(* Logix 5000 project; controller ARS14002_PLC vendor 1 type 14 code 218 rev 30.11; software revision 30.01; part 10 of 13 *)
(* tags used below, declared in another part *)
   DERIME_EMPTY : BOOL;
   DERIME_EMPTY_ALARM : BOOL;
   DERIME_EMPTY_HOLD_TMR : TIMER;
   DERIME_FILL : BOOL;
   DERIME_FULL : BOOL;
   DERIME_FULL_ALARM : BOOL;
   DERIME_FULL_HOLD_TMR : TIMER;
   DERIME_SPH : REAL;
   DERIME_SPL : REAL;
   DERIME_VENT : BOOL;
   ARS_DERIME_AUTO : BOOL;
   AT2_PLANT_ATOMIZING : BOOL;
   AT3_PLANT_ATOMIZING : BOOL;
   BLOWBACK_PRESS_SPH : REAL;
   BLOWBACK_PRESS_SPL : REAL;
   BLOWBACK_PRESS_UNSAFE : REAL;
   DERIME_HOLD : BOOL;
   DERIME_HP_CYCLE : BOOL;
   DERIME_HP_SPH : REAL;   // SETPOINT FOR VALVES BESIDES FCV-202
   DERIME_HP_SPL : REAL;   // SETPOIT FOR VALVES BESIDES FCV-202
   FCV_202 : CM_AO_VLV;
   FCV_202_BLOWBACK_POS : REAL;
   FCV_504_SP_Standby : REAL;
   FCV_504_SP_Standby_AR : REAL;
   FCV_504_SP_Standby_FRONT_END : REAL;
   FIRST_SCAN_BIT : BOOL;
   FVR_800C_RUNNING : BOOL;
   FVR_800D_RUNNING : BOOL;
   MTR_550 : CM_DO_FVNR;
   PDT_1101A : CM_AI_SCL_ALT;
   PIDE_101A : PID_ENHANCED;
   PIDE_101B : PID_ENHANCED;
   PIDE_101C : PID_ENHANCED;
   PIDE_102A : PID_ENHANCED;
   PIDE_102B : PID_ENHANCED;
   PIDE_102C : PID_ENHANCED;
   PIDE_202 : PID_ENHANCED;
   PIDE_204 : PID_ENHANCED;
   PIDE_207 : PID_ENHANCED;
   PIDE_504 : PID_ENHANCED;
   PIDE_504_COLDBOX_IGAIN : REAL;
   PIDE_504_COLDBOX_PGAIN : REAL;
   PIDE_504_FRONT_END_CONTROL : BOOL;
   PIDE_504_FRONT_END_IGAIN : REAL;
   PIDE_504_FRONT_END_PGAIN : REAL;
   PIDE_504_MODE : BOOL;   // 0 = Argon (PT-601) 1 = N2 (PT-603)
   PIDE_504_PVCHANGE1 : BOOL;
   PIDE_504_PVCHANGE2 : BOOL;
   PIDE_504_PVCHANGE3 : BOOL;
   PIDE_504_RESET : BOOL;
   PIDE_603 : PID_ENHANCED;
   PILOT_PLANT_ATOMIZING : BOOL;
   PT_1003 : CM_AI_SCL;
   PT_1101A : CM_AI_SCL;
   PT_1301A : CM_AI_SCL;
   PT_1301B : CM_AI_SCL;
   PT_201 : CM_AI_SCL;
   PT_601 : CM_AI_SCL;
   PT_603 : CM_AI_SCL;
   PT_701 : CM_AI_SCL;
   PT_806 : CM_AI_SCL;
   PWHMI_OutletValveStatus : BOOL;
   SV_1005_SPH : INT;
   SV_1005_SPL : INT;
   SV_1005X : CM_DO_GENERIC;
   SV_101AF : CM_DO_GENERIC;
   SV_101BF : CM_DO_GENERIC;
   SV_101CF : CM_DO_GENERIC;
   SV_102AF : CM_DO_GENERIC;
   SV_102BF : CM_DO_GENERIC;
   SV_102CF : CM_DO_GENERIC;
   SV_1104A : CM_DO_GENERIC;
   SV_1109AX : CM_DO_GENERIC;
   SV_1304A : CM_DO_GENERIC;
   SV_1304B : CM_DO_GENERIC;
   SV_1309AX : CM_DO_GENERIC;
   SV_1309BX : CM_DO_GENERIC;
   SV_202F : CM_DO_GENERIC;
   SV_204F : CM_DO_GENERIC;
   SV_207F : CM_DO_GENERIC;
   SV_504F : CM_DO_GENERIC;
   TK_1100A_Low : BOOL;
   TK_1100A_LOW_DLA_TMR : TIMER;
   TK_1100A_Low_SPH : REAL;
   TK_1100A_Low_SPL : REAL;
   TK_1100A_Low_Warning : BOOL;
   TK_1100A_LOW_WARNING_DLA_TMR : TIMER;
   TK_1100A_Low_WARNING_SPH : REAL;
   TK_1100A_Low_WARNING_SPL : REAL;
   TK_1100A_PBC_Pressure_SPH : INT;
   TK_1100A_PBC_Pressure_SPL : INT;
   TK_1100A_Vent_Closed_TMR : TIMER;
   TK_1100A_Vent_Open_TMR : TIMER;
   TK_1100A_Vent_Pressure_SPH : INT;
   TK_1100A_Vent_Pressure_SPL : INT;
   TK_1300A_PBC_Pressure_SPH : INT;
   TK_1300A_PBC_Pressure_SPL : INT;
   TK_1300A_Vent_Closed_TMR : TIMER;
   TK_1300A_Vent_Open_TMR : TIMER;
   TK_1300A_Vent_Pressure_SPH : INT;
   TK_1300A_Vent_Pressure_SPL : INT;
   TK_1300B_Vent_Closed_TMR : TIMER;
   TK_1300B_Vent_Open_TMR : TIMER;
   XV_623 : CM_DO_VLV;
   XV_623_FILL_MODE : BOOL;   // (0=Manual, 1=Auto)
   XV_623_SPH : INT;
   XV_623_SPL : INT;
   XV_801A : CM_DO_VLV;
   XV_801B : CM_DO_VLV;
   XV_801C : CM_DO_VLV;
   XV_801D : CM_DO_VLV;
   XV_806 : CM_DO_VLV;
(* MainProgram, continued *)

ROUTINE _310_TK_1100A   (* ladder *)
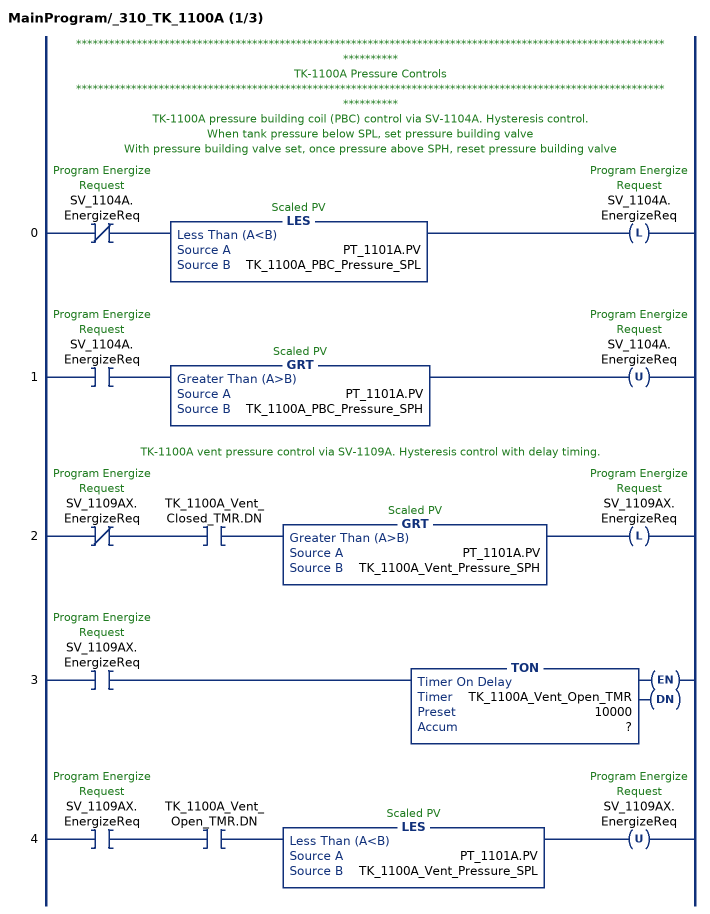
   // *********************************************************************************************************************
   // TK-1100A Pressure Controls
   // *********************************************************************************************************************
   // TK-1100A pressure building coil (PBC) control via SV-1104A. Hysteresis control.
   // When tank pressure below SPL, set pressure building valve
   // With pressure building valve set, once pressure above SPH, reset pressure building valve
   0: XIO(SV_1104A.EnergizeReq)LES(PT_1101A.PV,TK_1100A_PBC_Pressure_SPL)OTL(SV_1104A.EnergizeReq);
   1: XIC(SV_1104A.EnergizeReq)GRT(PT_1101A.PV,TK_1100A_PBC_Pressure_SPH)OTU(SV_1104A.EnergizeReq);
   // TK-1100A vent pressure control via SV-1109A. Hysteresis control with delay timing.
   2: XIO(SV_1109AX.EnergizeReq)XIC(TK_1100A_Vent_Closed_TMR.DN)GRT(PT_1101A.PV,TK_1100A_Vent_Pressure_SPH)OTL(SV_1109AX.EnergizeReq);
   3: XIC(SV_1109AX.EnergizeReq)TON(TK_1100A_Vent_Open_TMR,?,?);
   4: XIC(SV_1109AX.EnergizeReq)XIC(TK_1100A_Vent_Open_TMR.DN)LES(PT_1101A.PV,TK_1100A_Vent_Pressure_SPL)OTU(SV_1109AX.EnergizeReq);
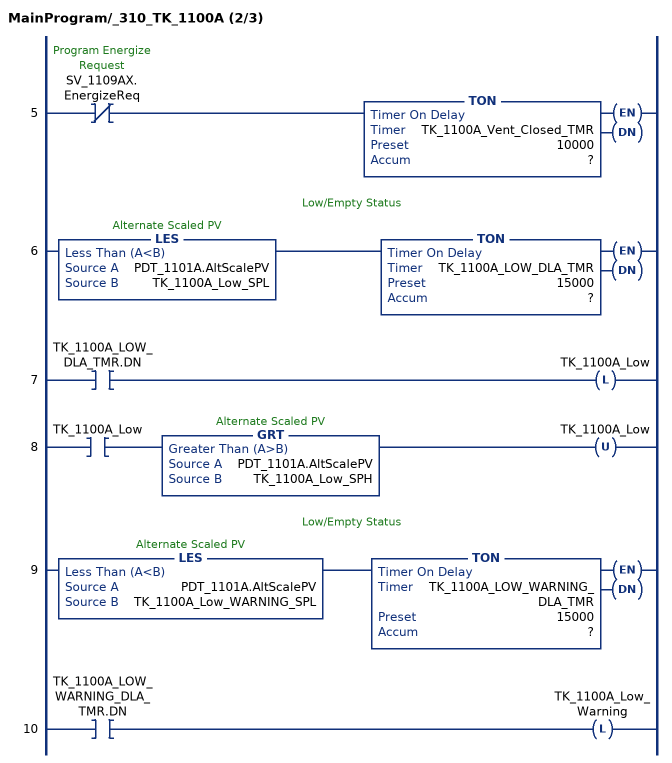
   5: XIO(SV_1109AX.EnergizeReq)TON(TK_1100A_Vent_Closed_TMR,?,?);
   // Low/Empty Status
   6: LES(PDT_1101A.AltScalePV,TK_1100A_Low_SPL)TON(TK_1100A_LOW_DLA_TMR,?,?);
   7: XIC(TK_1100A_LOW_DLA_TMR.DN)OTL(TK_1100A_Low);
   8: XIC(TK_1100A_Low)GRT(PDT_1101A.AltScalePV,TK_1100A_Low_SPH)OTU(TK_1100A_Low);
   // Low/Empty Status
   9: LES(PDT_1101A.AltScalePV,TK_1100A_Low_WARNING_SPL)TON(TK_1100A_LOW_WARNING_DLA_TMR,?,?);
   10: XIC(TK_1100A_LOW_WARNING_DLA_TMR.DN)OTL(TK_1100A_Low_Warning);
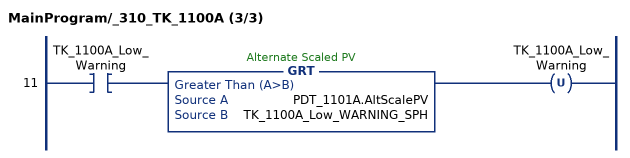
   11: XIC(TK_1100A_Low_Warning)GRT(PDT_1101A.AltScalePV,TK_1100A_Low_WARNING_SPH)OTU(TK_1100A_Low_Warning);
END_ROUTINE

ROUTINE _311A_TK_1300A   (* ladder *)
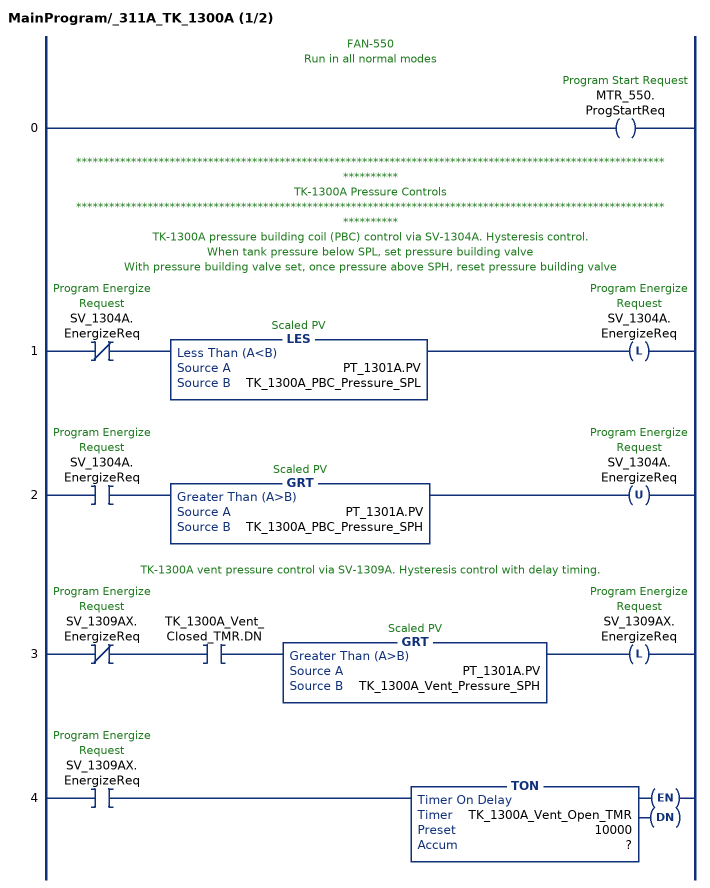
   // FAN-550
   // Run in all normal modes
   0: OTE(MTR_550.ProgStartReq);
   // *********************************************************************************************************************
   // TK-1300A Pressure Controls
   // *********************************************************************************************************************
   // TK-1300A pressure building coil (PBC) control via SV-1304A. Hysteresis control.
   // When tank pressure below SPL, set pressure building valve
   // With pressure building valve set, once pressure above SPH, reset pressure building valve
   1: XIO(SV_1304A.EnergizeReq)LES(PT_1301A.PV,TK_1300A_PBC_Pressure_SPL)OTL(SV_1304A.EnergizeReq);
   2: XIC(SV_1304A.EnergizeReq)GRT(PT_1301A.PV,TK_1300A_PBC_Pressure_SPH)OTU(SV_1304A.EnergizeReq);
   // TK-1300A vent pressure control via SV-1309A. Hysteresis control with delay timing.
   3: XIO(SV_1309AX.EnergizeReq)XIC(TK_1300A_Vent_Closed_TMR.DN)GRT(PT_1301A.PV,TK_1300A_Vent_Pressure_SPH)OTL(SV_1309AX.EnergizeReq);
   4: XIC(SV_1309AX.EnergizeReq)TON(TK_1300A_Vent_Open_TMR,?,?);
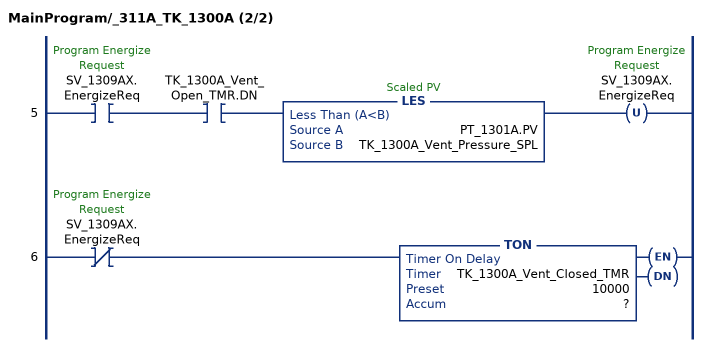
   5: XIC(SV_1309AX.EnergizeReq)XIC(TK_1300A_Vent_Open_TMR.DN)LES(PT_1301A.PV,TK_1300A_Vent_Pressure_SPL)OTU(SV_1309AX.EnergizeReq);
   6: XIO(SV_1309AX.EnergizeReq)TON(TK_1300A_Vent_Closed_TMR,?,?);
END_ROUTINE

ROUTINE _311B_TK_1300B   (* ladder *)
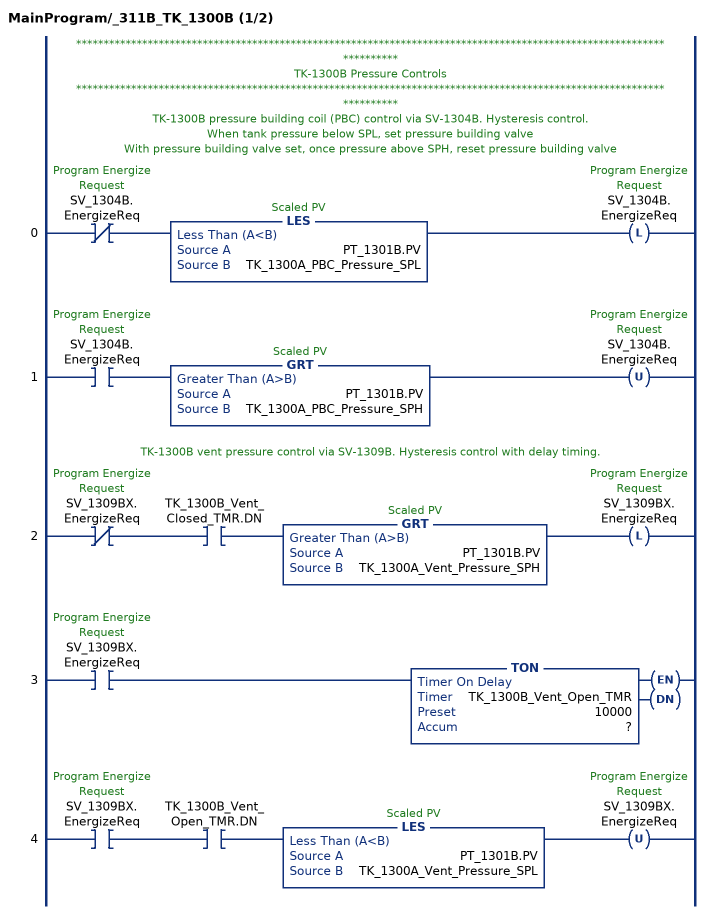
   // *********************************************************************************************************************
   // TK-1300B Pressure Controls
   // *********************************************************************************************************************
   // TK-1300B pressure building coil (PBC) control via SV-1304B. Hysteresis control.
   // When tank pressure below SPL, set pressure building valve
   // With pressure building valve set, once pressure above SPH, reset pressure building valve
   0: XIO(SV_1304B.EnergizeReq)LES(PT_1301B.PV,TK_1300A_PBC_Pressure_SPL)OTL(SV_1304B.EnergizeReq);
   1: XIC(SV_1304B.EnergizeReq)GRT(PT_1301B.PV,TK_1300A_PBC_Pressure_SPH)OTU(SV_1304B.EnergizeReq);
   // TK-1300B vent pressure control via SV-1309B. Hysteresis control with delay timing.
   2: XIO(SV_1309BX.EnergizeReq)XIC(TK_1300B_Vent_Closed_TMR.DN)GRT(PT_1301B.PV,TK_1300A_Vent_Pressure_SPH)OTL(SV_1309BX.EnergizeReq);
   3: XIC(SV_1309BX.EnergizeReq)TON(TK_1300B_Vent_Open_TMR,?,?);
   4: XIC(SV_1309BX.EnergizeReq)XIC(TK_1300B_Vent_Open_TMR.DN)LES(PT_1301B.PV,TK_1300A_Vent_Pressure_SPL)OTU(SV_1309BX.EnergizeReq);
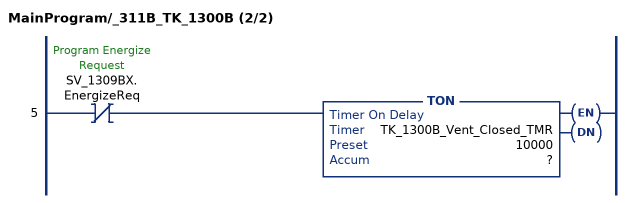
   5: XIO(SV_1309BX.EnergizeReq)TON(TK_1300B_Vent_Closed_TMR,?,?);
END_ROUTINE

ROUTINE _312_Misc_Hysteresis   (* ladder *)
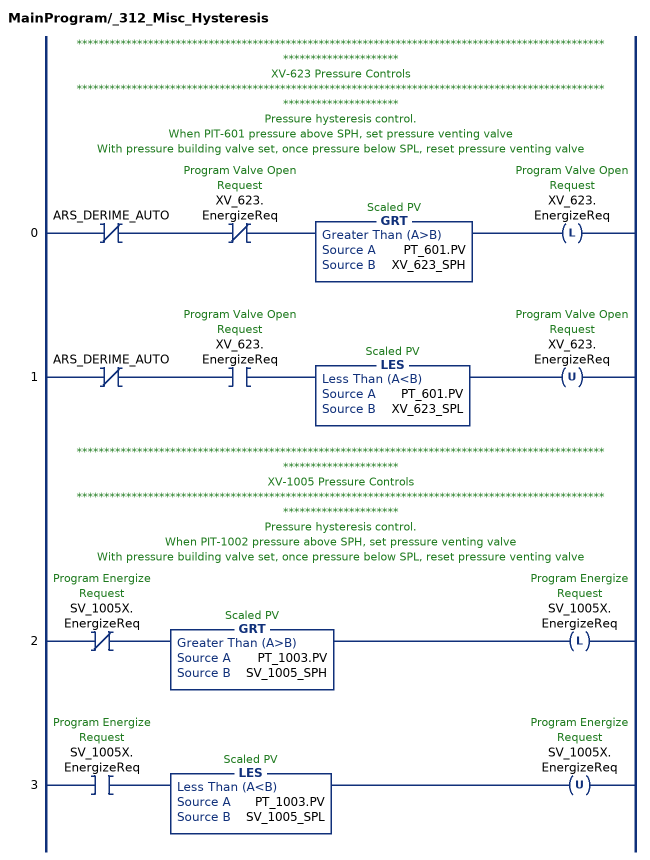
   // *********************************************************************************************************************
   // XV-623 Pressure Controls
   // *********************************************************************************************************************
   // Pressure hysteresis control.
   // When PIT-601 pressure above SPH, set pressure venting valve
   // With pressure building valve set, once pressure below SPL, reset pressure venting valve
   0: XIO(ARS_DERIME_AUTO)XIO(XV_623.EnergizeReq)GRT(PT_601.PV,XV_623_SPH)OTL(XV_623.EnergizeReq);
   1: XIO(ARS_DERIME_AUTO)XIC(XV_623.EnergizeReq)LES(PT_601.PV,XV_623_SPL)OTU(XV_623.EnergizeReq);
   // *********************************************************************************************************************
   // XV-1005 Pressure Controls
   // *********************************************************************************************************************
   // Pressure hysteresis control.
   // When PIT-1002 pressure above SPH, set pressure venting valve
   // With pressure building valve set, once pressure below SPL, reset pressure venting valve
   2: XIO(SV_1005X.EnergizeReq)GRT(PT_1003.PV,SV_1005_SPH)OTL(SV_1005X.EnergizeReq);
   3: XIC(SV_1005X.EnergizeReq)LES(PT_1003.PV,SV_1005_SPL)OTU(SV_1005X.EnergizeReq);
END_ROUTINE

ROUTINE _313_Derime   (* ladder *)
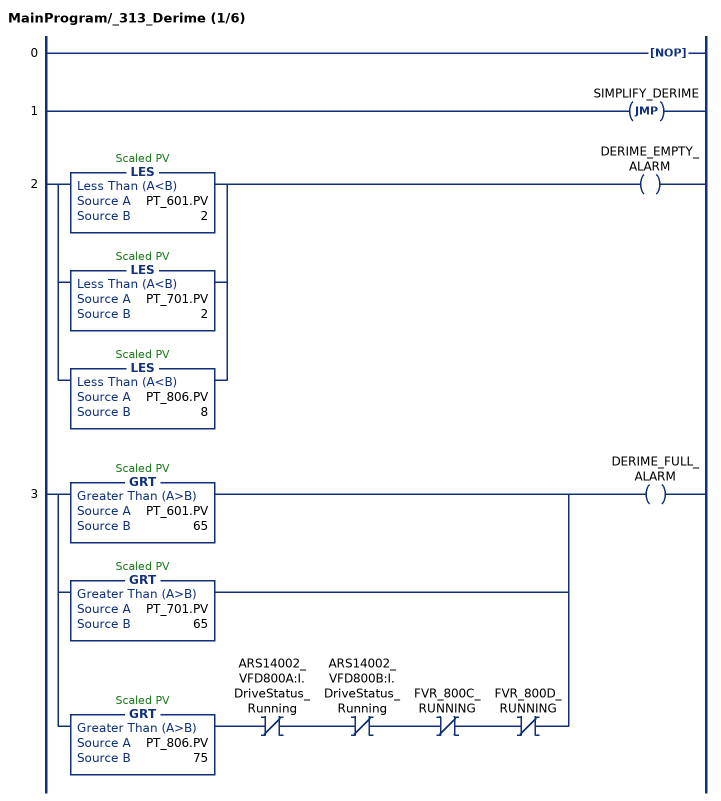
   0: NOP();
   1: JMP(SIMPLIFY_DERIME);
   2: [LES(PT_601.PV,2) ,LES(PT_701.PV,2) ,LES(PT_806.PV,8) ]OTE(DERIME_EMPTY_ALARM);
   3: [GRT(PT_601.PV,65) ,GRT(PT_701.PV,65) ,GRT(PT_806.PV,75) XIO(ARS14002_VFD800A:I.DriveStatus_Running) XIO(ARS14002_VFD800B:I.DriveStatus_Running) XIO(FVR_800C_RUNNING) XIO(FVR_800D_RUNNING) ]OTE(DERIME_FULL_ALARM);
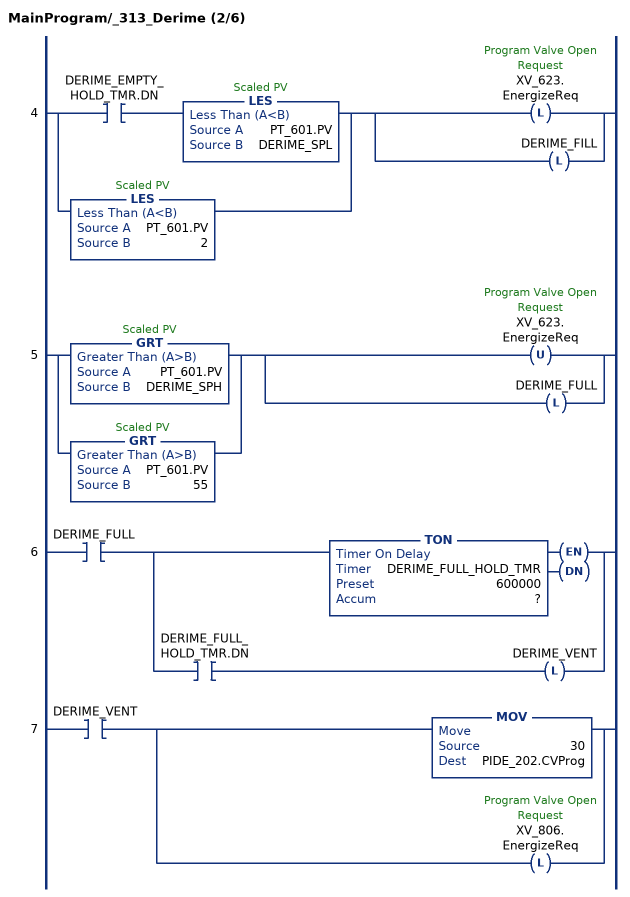
   4: [XIC(DERIME_EMPTY_HOLD_TMR.DN) LES(PT_601.PV,DERIME_SPL) ,LES(PT_601.PV,2) ][OTL(XV_623.EnergizeReq) ,OTL(DERIME_FILL) ];
   5: [GRT(PT_601.PV,DERIME_SPH) ,GRT(PT_601.PV,55) ][OTU(XV_623.EnergizeReq) ,OTL(DERIME_FULL) ];
   6: XIC(DERIME_FULL)[TON(DERIME_FULL_HOLD_TMR,?,?) ,XIC(DERIME_FULL_HOLD_TMR.DN) OTL(DERIME_VENT) ];
   7: XIC(DERIME_VENT)[MOV(30,PIDE_202.CVProg) ,OTL(XV_806.EnergizeReq) ];
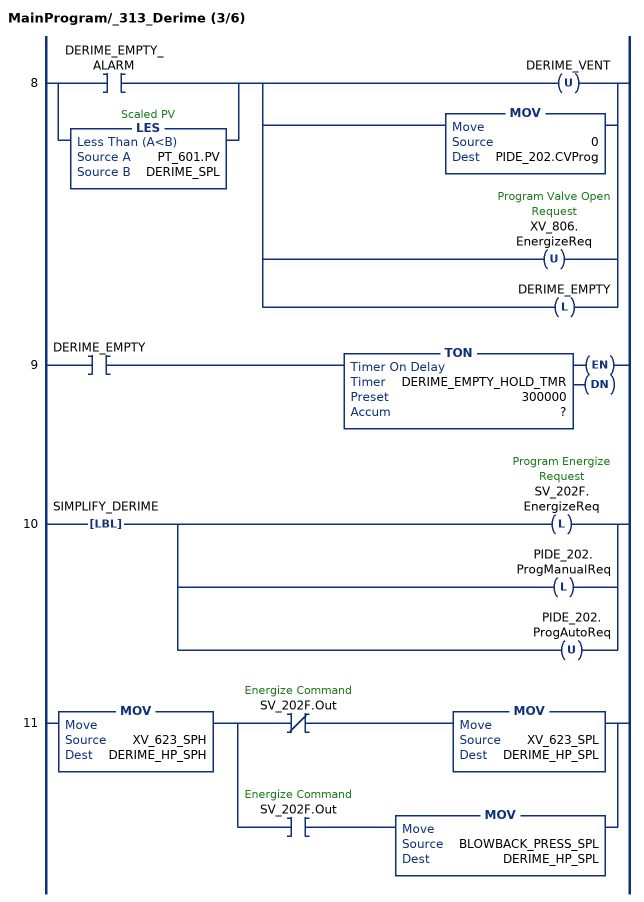
   8: [XIC(DERIME_EMPTY_ALARM) ,LES(PT_601.PV,DERIME_SPL) ][OTU(DERIME_VENT) ,MOV(0,PIDE_202.CVProg) ,OTU(XV_806.EnergizeReq) ,OTL(DERIME_EMPTY) ];
   9: XIC(DERIME_EMPTY)TON(DERIME_EMPTY_HOLD_TMR,?,?);
   10: LBL(SIMPLIFY_DERIME)[OTL(SV_202F.EnergizeReq) ,OTL(PIDE_202.ProgManualReq) ,OTU(PIDE_202.ProgAutoReq) ];
   11: MOV(XV_623_SPH,DERIME_HP_SPH)[XIO(SV_202F.Out) MOV(XV_623_SPL,DERIME_HP_SPL) ,XIC(SV_202F.Out) MOV(BLOWBACK_PRESS_SPL,DERIME_HP_SPL) ];
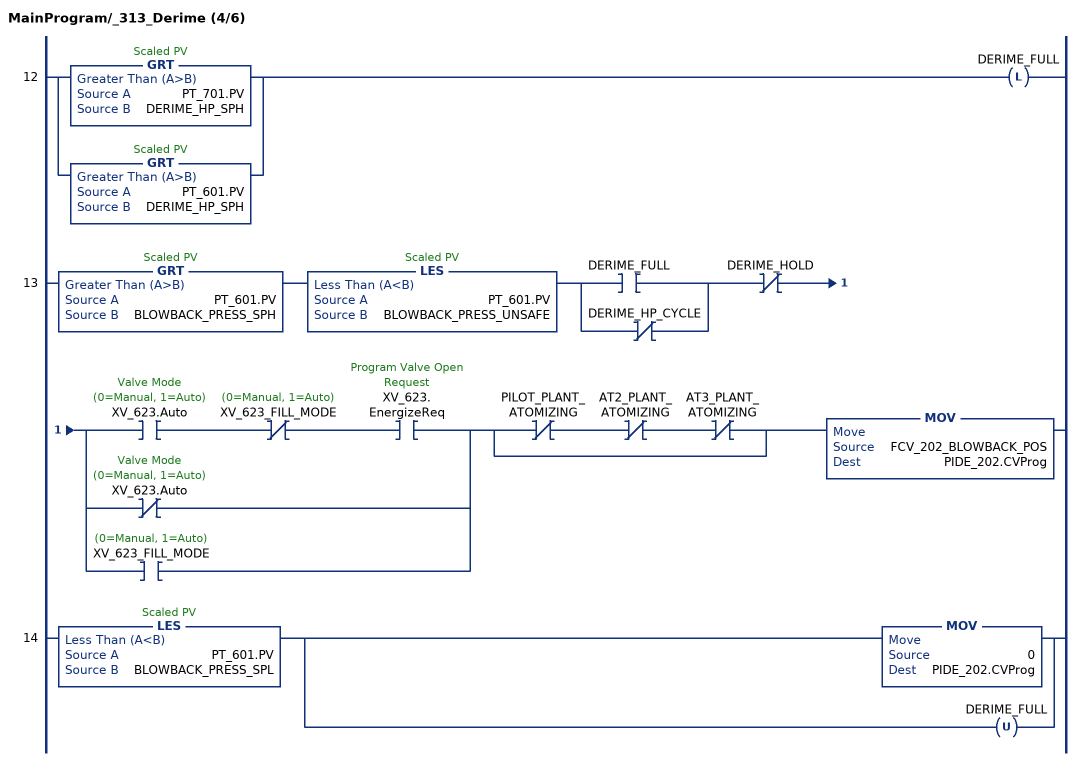
   12: [GRT(PT_701.PV,DERIME_HP_SPH) ,GRT(PT_601.PV,DERIME_HP_SPH) ]OTL(DERIME_FULL);
   13: GRT(PT_601.PV,BLOWBACK_PRESS_SPH)LES(PT_601.PV,BLOWBACK_PRESS_UNSAFE)[XIC(DERIME_FULL) ,XIO(DERIME_HP_CYCLE) ]XIO(DERIME_HOLD)[XIC(XV_623.Auto) XIO(XV_623_FILL_MODE) XIC(XV_623.EnergizeReq) ,XIO(XV_623.Auto) ,XIC(XV_623_FILL_MODE) ][XIO(PILOT_PLANT_ATOMIZING) XIO(AT2_PLANT_ATOMIZING) XIO(AT3_PLANT_ATOMIZING) ,]MOV(FCV_202_BLOWBACK_POS,PIDE_202.CVProg);
   14: LES(PT_601.PV,BLOWBACK_PRESS_SPL)[MOV(0,PIDE_202.CVProg) ,OTU(DERIME_FULL) ];
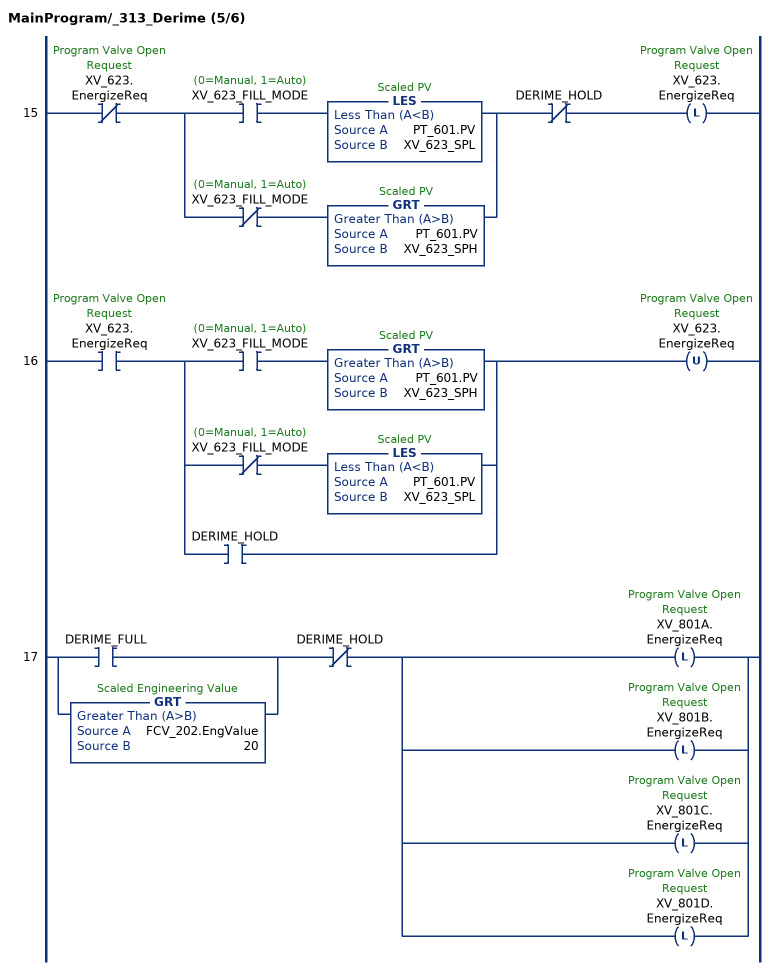
   15: XIO(XV_623.EnergizeReq)[XIC(XV_623_FILL_MODE) LES(PT_601.PV,XV_623_SPL) ,XIO(XV_623_FILL_MODE) GRT(PT_601.PV,XV_623_SPH) ]XIO(DERIME_HOLD)OTL(XV_623.EnergizeReq);
   16: XIC(XV_623.EnergizeReq)[XIC(XV_623_FILL_MODE) GRT(PT_601.PV,XV_623_SPH) ,XIO(XV_623_FILL_MODE) LES(PT_601.PV,XV_623_SPL) ,XIC(DERIME_HOLD) ]OTU(XV_623.EnergizeReq);
   17: [XIC(DERIME_FULL) ,GRT(FCV_202.EngValue,20) ]XIO(DERIME_HOLD)[OTL(XV_801A.EnergizeReq) ,OTL(XV_801B.EnergizeReq) ,OTL(XV_801C.EnergizeReq) ,OTL(XV_801D.EnergizeReq) ];
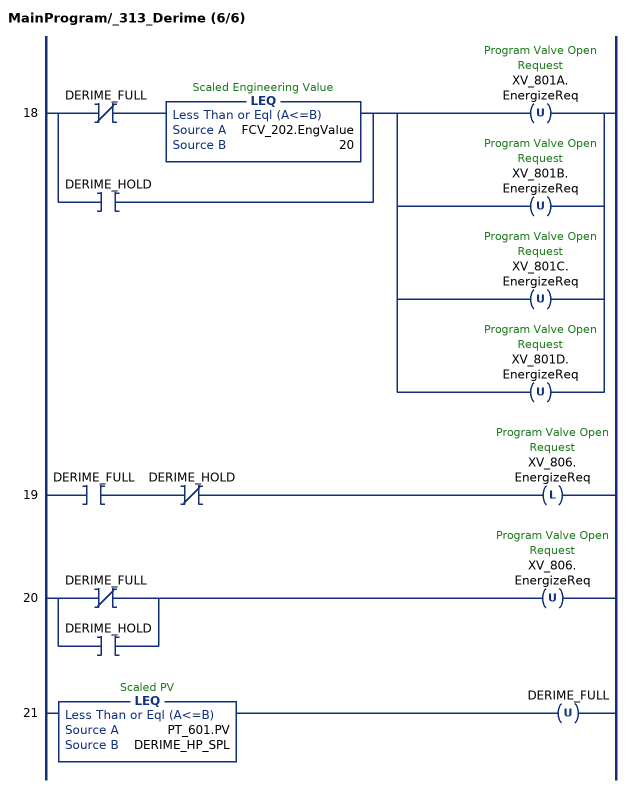
   18: [XIO(DERIME_FULL) LEQ(FCV_202.EngValue,20) ,XIC(DERIME_HOLD) ][OTU(XV_801A.EnergizeReq) ,OTU(XV_801B.EnergizeReq) ,OTU(XV_801C.EnergizeReq) ,OTU(XV_801D.EnergizeReq) ];
   19: XIC(DERIME_FULL)XIO(DERIME_HOLD)OTL(XV_806.EnergizeReq);
   20: [XIO(DERIME_FULL) ,XIC(DERIME_HOLD) ]OTU(XV_806.EnergizeReq);
   21: LEQ(PT_601.PV,DERIME_HP_SPL)OTU(DERIME_FULL);
END_ROUTINE

ROUTINE _40_Process_PID_Misc   (* ladder *)
// PID state transition logic
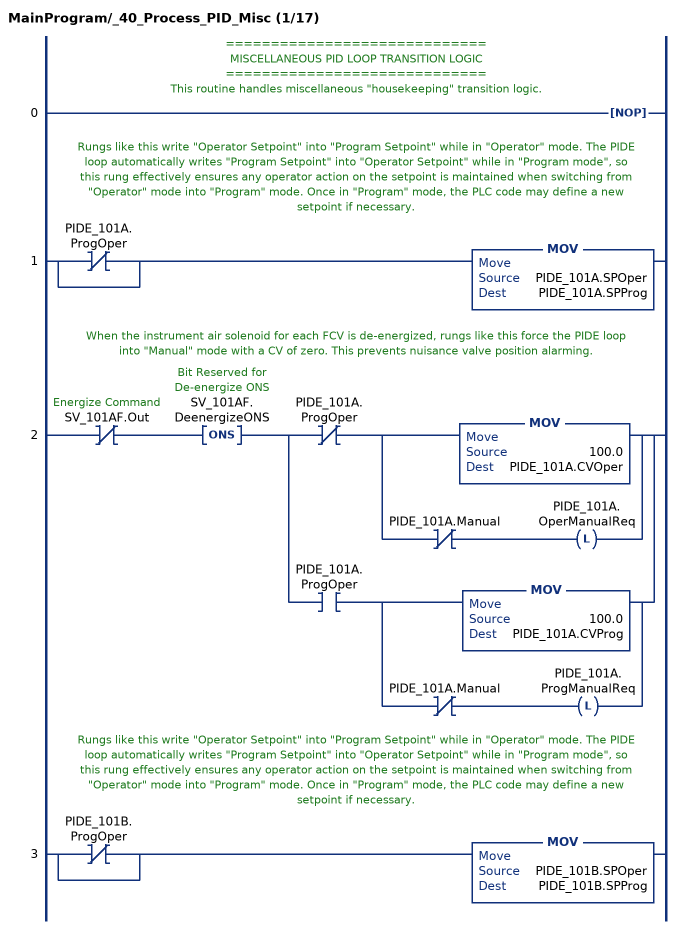
   // =============================
   // MISCELLANEOUS PID LOOP TRANSITION LOGIC
   // =============================
   //  This routine handles miscellaneous "housekeeping" transition logic.
   0: NOP();
   // Rungs like this write "Operator Setpoint" into "Program Setpoint" while in "Operator" mode. The PIDE loop automatically writes "Program Setpoint" into "Operator Setpoint" while in "Program mode", so this rung effectively ensures any operator action on the setpoint is maintained when switching from "Operator" mode into "Program" mode. Once in "Program" mode, the PLC code may define a new setpoint if necessary.
   1: [XIO(PIDE_101A.ProgOper) ,]MOV(PIDE_101A.SPOper,PIDE_101A.SPProg);
   // When the instrument air solenoid for each FCV is de-energized, rungs like this force the PIDE loop into "Manual" mode with a CV of zero. This prevents nuisance valve position alarming.
   2: XIO(SV_101AF.Out)ONS(SV_101AF.DeenergizeONS)[XIO(PIDE_101A.ProgOper) [MOV(100.0,PIDE_101A.CVOper) ,XIO(PIDE_101A.Manual) OTL(PIDE_101A.OperManualReq) ] ,XIC(PIDE_101A.ProgOper) [MOV(100.0,PIDE_101A.CVProg) ,XIO(PIDE_101A.Manual) OTL(PIDE_101A.ProgManualReq) ] ];
   // Rungs like this write "Operator Setpoint" into "Program Setpoint" while in "Operator" mode. The PIDE loop automatically writes "Program Setpoint" into "Operator Setpoint" while in "Program mode", so this rung effectively ensures any operator action on the setpoint is maintained when switching from "Operator" mode into "Program" mode. Once in "Program" mode, the PLC code may define a new setpoint if necessary.
   3: [XIO(PIDE_101B.ProgOper) ,]MOV(PIDE_101B.SPOper,PIDE_101B.SPProg);
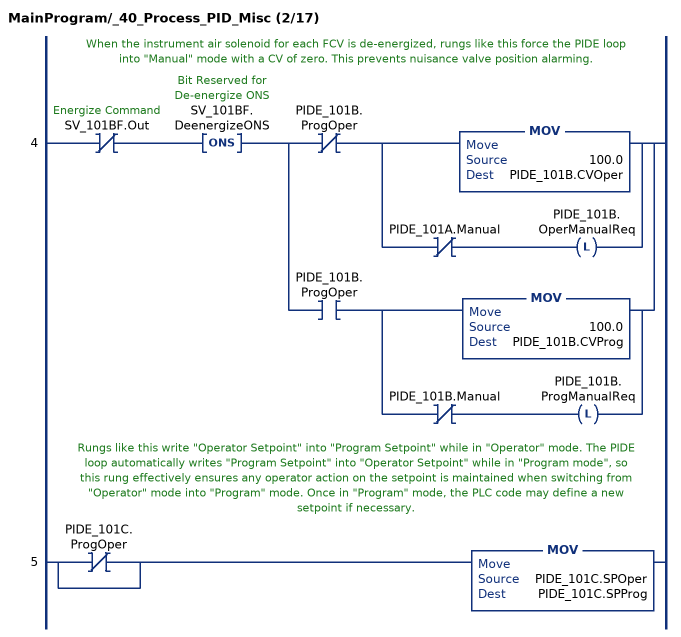
   // When the instrument air solenoid for each FCV is de-energized, rungs like this force the PIDE loop into "Manual" mode with a CV of zero. This prevents nuisance valve position alarming.
   4: XIO(SV_101BF.Out)ONS(SV_101BF.DeenergizeONS)[XIO(PIDE_101B.ProgOper) [MOV(100.0,PIDE_101B.CVOper) ,XIO(PIDE_101A.Manual) OTL(PIDE_101B.OperManualReq) ] ,XIC(PIDE_101B.ProgOper) [MOV(100.0,PIDE_101B.CVProg) ,XIO(PIDE_101B.Manual) OTL(PIDE_101B.ProgManualReq) ] ];
   // Rungs like this write "Operator Setpoint" into "Program Setpoint" while in "Operator" mode. The PIDE loop automatically writes "Program Setpoint" into "Operator Setpoint" while in "Program mode", so this rung effectively ensures any operator action on the setpoint is maintained when switching from "Operator" mode into "Program" mode. Once in "Program" mode, the PLC code may define a new setpoint if necessary.
   5: [XIO(PIDE_101C.ProgOper) ,]MOV(PIDE_101C.SPOper,PIDE_101C.SPProg);
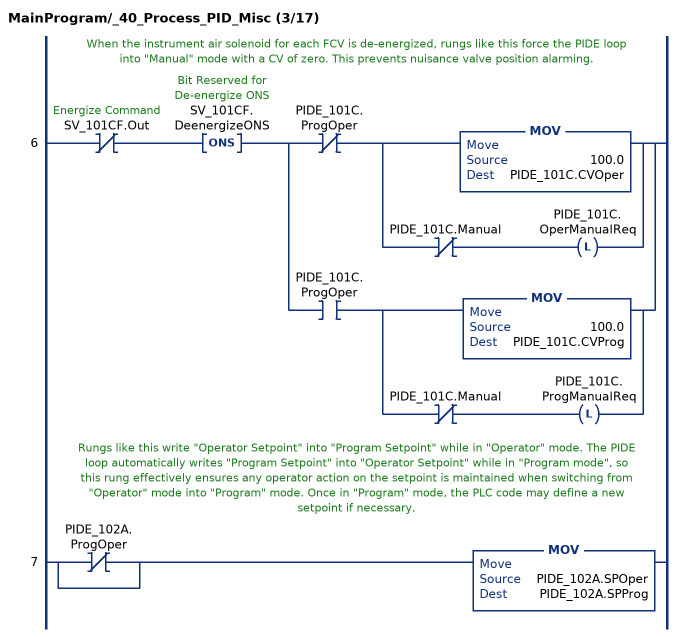
   // When the instrument air solenoid for each FCV is de-energized, rungs like this force the PIDE loop into "Manual" mode with a CV of zero. This prevents nuisance valve position alarming.
   6: XIO(SV_101CF.Out)ONS(SV_101CF.DeenergizeONS)[XIO(PIDE_101C.ProgOper) [MOV(100.0,PIDE_101C.CVOper) ,XIO(PIDE_101C.Manual) OTL(PIDE_101C.OperManualReq) ] ,XIC(PIDE_101C.ProgOper) [MOV(100.0,PIDE_101C.CVProg) ,XIO(PIDE_101C.Manual) OTL(PIDE_101C.ProgManualReq) ] ];
   // Rungs like this write "Operator Setpoint" into "Program Setpoint" while in "Operator" mode. The PIDE loop automatically writes "Program Setpoint" into "Operator Setpoint" while in "Program mode", so this rung effectively ensures any operator action on the setpoint is maintained when switching from "Operator" mode into "Program" mode. Once in "Program" mode, the PLC code may define a new setpoint if necessary.
   7: [XIO(PIDE_102A.ProgOper) ,]MOV(PIDE_102A.SPOper,PIDE_102A.SPProg);
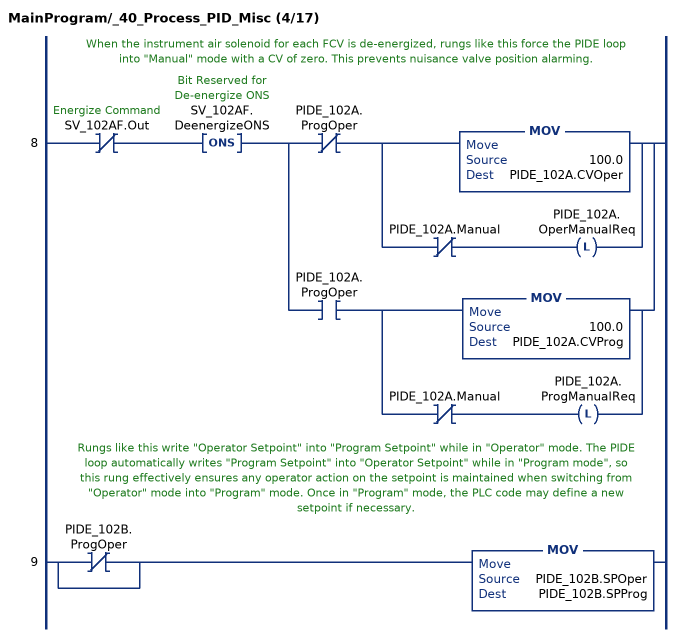
   // When the instrument air solenoid for each FCV is de-energized, rungs like this force the PIDE loop into "Manual" mode with a CV of zero. This prevents nuisance valve position alarming.
   8: XIO(SV_102AF.Out)ONS(SV_102AF.DeenergizeONS)[XIO(PIDE_102A.ProgOper) [MOV(100.0,PIDE_102A.CVOper) ,XIO(PIDE_102A.Manual) OTL(PIDE_102A.OperManualReq) ] ,XIC(PIDE_102A.ProgOper) [MOV(100.0,PIDE_102A.CVProg) ,XIO(PIDE_102A.Manual) OTL(PIDE_102A.ProgManualReq) ] ];
   // Rungs like this write "Operator Setpoint" into "Program Setpoint" while in "Operator" mode. The PIDE loop automatically writes "Program Setpoint" into "Operator Setpoint" while in "Program mode", so this rung effectively ensures any operator action on the setpoint is maintained when switching from "Operator" mode into "Program" mode. Once in "Program" mode, the PLC code may define a new setpoint if necessary.
   9: [XIO(PIDE_102B.ProgOper) ,]MOV(PIDE_102B.SPOper,PIDE_102B.SPProg);
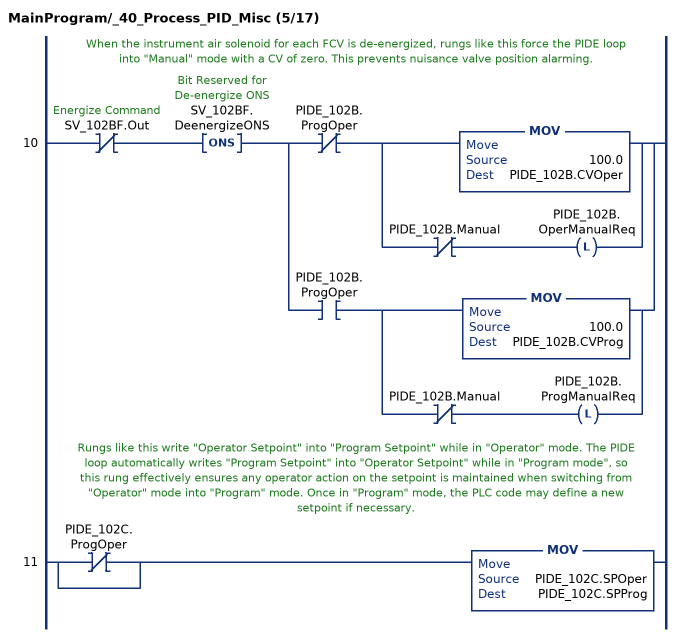
   // When the instrument air solenoid for each FCV is de-energized, rungs like this force the PIDE loop into "Manual" mode with a CV of zero. This prevents nuisance valve position alarming.
   10: XIO(SV_102BF.Out)ONS(SV_102BF.DeenergizeONS)[XIO(PIDE_102B.ProgOper) [MOV(100.0,PIDE_102B.CVOper) ,XIO(PIDE_102B.Manual) OTL(PIDE_102B.OperManualReq) ] ,XIC(PIDE_102B.ProgOper) [MOV(100.0,PIDE_102B.CVProg) ,XIO(PIDE_102B.Manual) OTL(PIDE_102B.ProgManualReq) ] ];
   // Rungs like this write "Operator Setpoint" into "Program Setpoint" while in "Operator" mode. The PIDE loop automatically writes "Program Setpoint" into "Operator Setpoint" while in "Program mode", so this rung effectively ensures any operator action on the setpoint is maintained when switching from "Operator" mode into "Program" mode. Once in "Program" mode, the PLC code may define a new setpoint if necessary.
   11: [XIO(PIDE_102C.ProgOper) ,]MOV(PIDE_102C.SPOper,PIDE_102C.SPProg);
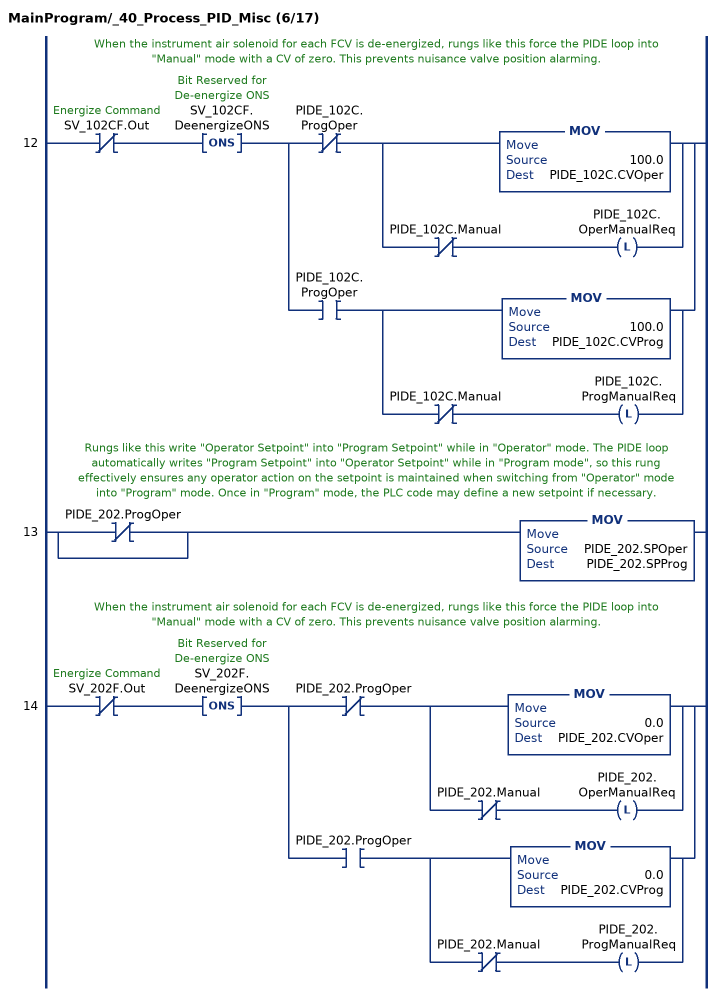
   // When the instrument air solenoid for each FCV is de-energized, rungs like this force the PIDE loop into "Manual" mode with a CV of zero. This prevents nuisance valve position alarming.
   12: XIO(SV_102CF.Out)ONS(SV_102CF.DeenergizeONS)[XIO(PIDE_102C.ProgOper) [MOV(100.0,PIDE_102C.CVOper) ,XIO(PIDE_102C.Manual) OTL(PIDE_102C.OperManualReq) ] ,XIC(PIDE_102C.ProgOper) [MOV(100.0,PIDE_102C.CVProg) ,XIO(PIDE_102C.Manual) OTL(PIDE_102C.ProgManualReq) ] ];
   // Rungs like this write "Operator Setpoint" into "Program Setpoint" while in "Operator" mode. The PIDE loop automatically writes "Program Setpoint" into "Operator Setpoint" while in "Program mode", so this rung effectively ensures any operator action on the setpoint is maintained when switching from "Operator" mode into "Program" mode. Once in "Program" mode, the PLC code may define a new setpoint if necessary.
   13: [XIO(PIDE_202.ProgOper) ,]MOV(PIDE_202.SPOper,PIDE_202.SPProg);
   // When the instrument air solenoid for each FCV is de-energized, rungs like this force the PIDE loop into "Manual" mode with a CV of zero. This prevents nuisance valve position alarming.
   14: XIO(SV_202F.Out)ONS(SV_202F.DeenergizeONS)[XIO(PIDE_202.ProgOper) [MOV(0.0,PIDE_202.CVOper) ,XIO(PIDE_202.Manual) OTL(PIDE_202.OperManualReq) ] ,XIC(PIDE_202.ProgOper) [MOV(0.0,PIDE_202.CVProg) ,XIO(PIDE_202.Manual) OTL(PIDE_202.ProgManualReq) ] ];
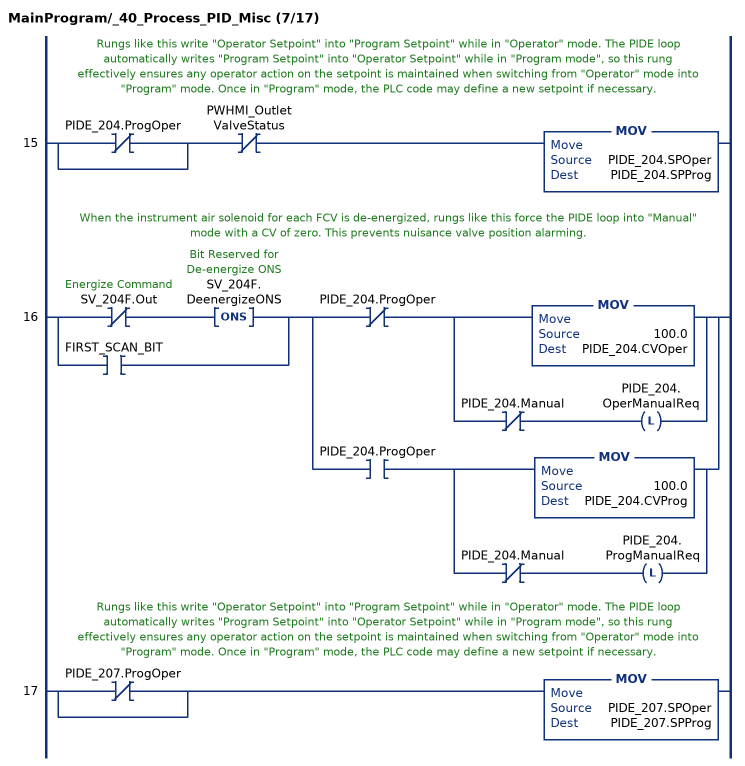
   // Rungs like this write "Operator Setpoint" into "Program Setpoint" while in "Operator" mode. The PIDE loop automatically writes "Program Setpoint" into "Operator Setpoint" while in "Program mode", so this rung effectively ensures any operator action on the setpoint is maintained when switching from "Operator" mode into "Program" mode. Once in "Program" mode, the PLC code may define a new setpoint if necessary.
   15: [XIO(PIDE_204.ProgOper) ,]XIO(PWHMI_OutletValveStatus)MOV(PIDE_204.SPOper,PIDE_204.SPProg);
   // When the instrument air solenoid for each FCV is de-energized, rungs like this force the PIDE loop into "Manual" mode with a CV of zero. This prevents nuisance valve position alarming.
   16: [XIO(SV_204F.Out) ONS(SV_204F.DeenergizeONS) ,XIC(FIRST_SCAN_BIT) ][XIO(PIDE_204.ProgOper) [MOV(100.0,PIDE_204.CVOper) ,XIO(PIDE_204.Manual) OTL(PIDE_204.OperManualReq) ] ,XIC(PIDE_204.ProgOper) [MOV(100.0,PIDE_204.CVProg) ,XIO(PIDE_204.Manual) OTL(PIDE_204.ProgManualReq) ] ];
   // Rungs like this write "Operator Setpoint" into "Program Setpoint" while in "Operator" mode. The PIDE loop automatically writes "Program Setpoint" into "Operator Setpoint" while in "Program mode", so this rung effectively ensures any operator action on the setpoint is maintained when switching from "Operator" mode into "Program" mode. Once in "Program" mode, the PLC code may define a new setpoint if necessary.
   17: [XIO(PIDE_207.ProgOper) ,]MOV(PIDE_207.SPOper,PIDE_207.SPProg);
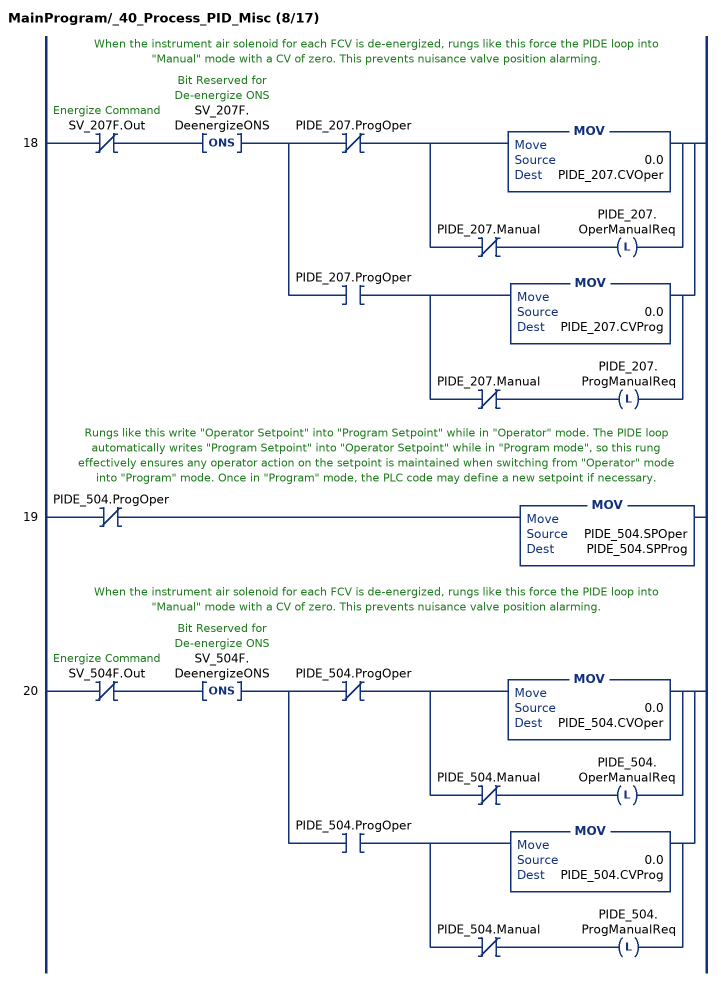
   // When the instrument air solenoid for each FCV is de-energized, rungs like this force the PIDE loop into "Manual" mode with a CV of zero. This prevents nuisance valve position alarming.
   18: XIO(SV_207F.Out)ONS(SV_207F.DeenergizeONS)[XIO(PIDE_207.ProgOper) [MOV(0.0,PIDE_207.CVOper) ,XIO(PIDE_207.Manual) OTL(PIDE_207.OperManualReq) ] ,XIC(PIDE_207.ProgOper) [MOV(0.0,PIDE_207.CVProg) ,XIO(PIDE_207.Manual) OTL(PIDE_207.ProgManualReq) ] ];
   // Rungs like this write "Operator Setpoint" into "Program Setpoint" while in "Operator" mode. The PIDE loop automatically writes "Program Setpoint" into "Operator Setpoint" while in "Program mode", so this rung effectively ensures any operator action on the setpoint is maintained when switching from "Operator" mode into "Program" mode. Once in "Program" mode, the PLC code may define a new setpoint if necessary.
   19: XIO(PIDE_504.ProgOper)MOV(PIDE_504.SPOper,PIDE_504.SPProg);
   // When the instrument air solenoid for each FCV is de-energized, rungs like this force the PIDE loop into "Manual" mode with a CV of zero. This prevents nuisance valve position alarming.
   20: XIO(SV_504F.Out)ONS(SV_504F.DeenergizeONS)[XIO(PIDE_504.ProgOper) [MOV(0.0,PIDE_504.CVOper) ,XIO(PIDE_504.Manual) OTL(PIDE_504.OperManualReq) ] ,XIC(PIDE_504.ProgOper) [MOV(0.0,PIDE_504.CVProg) ,XIO(PIDE_504.Manual) OTL(PIDE_504.ProgManualReq) ] ];
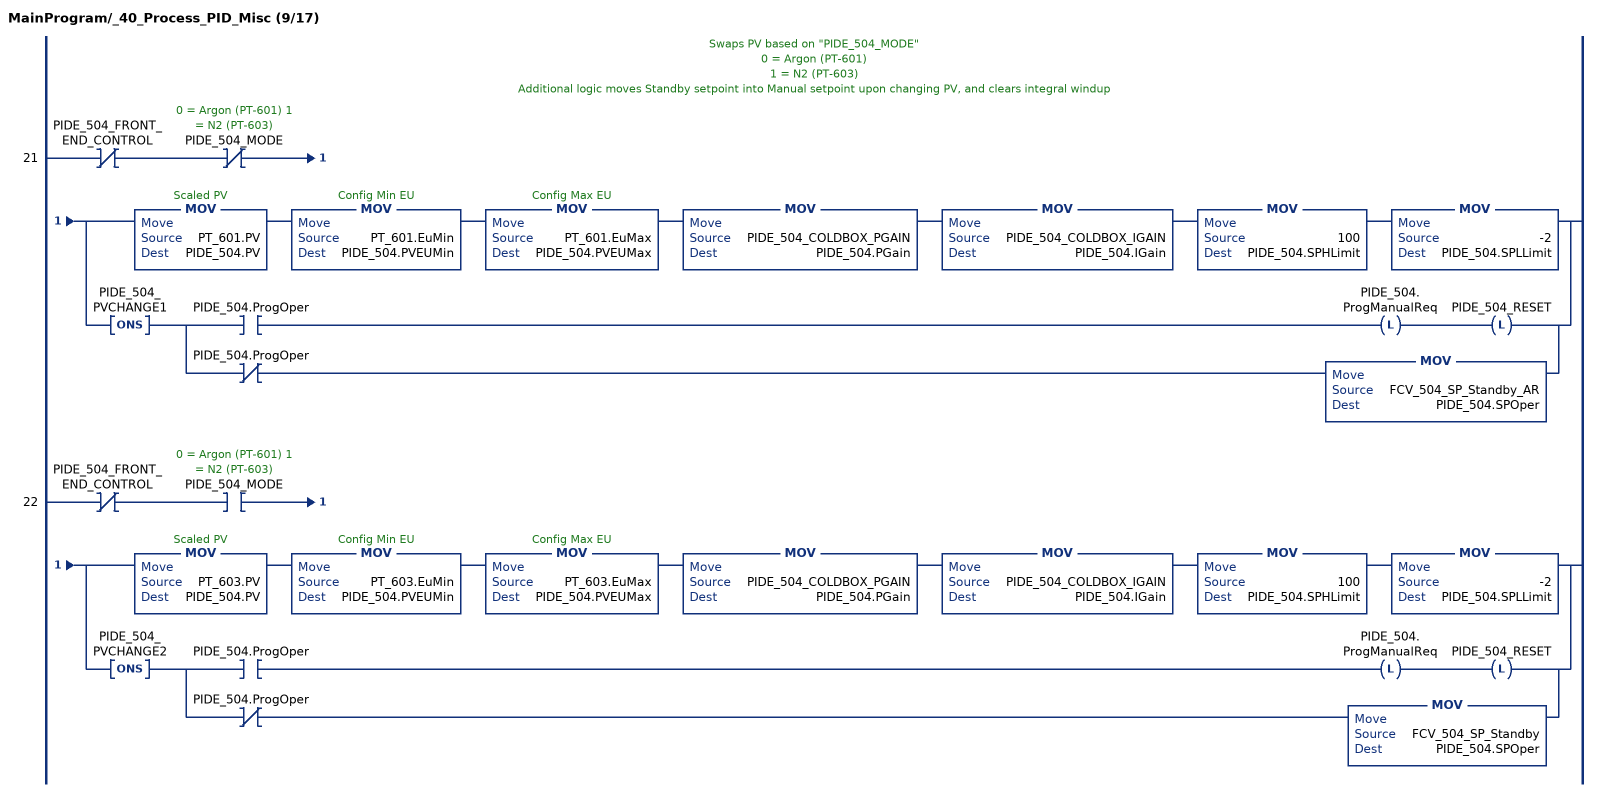
   // Swaps PV based on "PIDE_504_MODE"
   // 0 = Argon (PT-601)
   // 1 = N2 (PT-603)
   // Additional logic moves Standby setpoint into Manual setpoint upon changing PV, and clears integral windup
   21: XIO(PIDE_504_FRONT_END_CONTROL)XIO(PIDE_504_MODE)[MOV(PT_601.PV,PIDE_504.PV) MOV(PT_601.EuMin,PIDE_504.PVEUMin) MOV(PT_601.EuMax,PIDE_504.PVEUMax) MOV(PIDE_504_COLDBOX_PGAIN,PIDE_504.PGain) MOV(PIDE_504_COLDBOX_IGAIN,PIDE_504.IGain) MOV(100,PIDE_504.SPHLimit) MOV(-2,PIDE_504.SPLLimit) ,ONS(PIDE_504_PVCHANGE1) [XIC(PIDE_504.ProgOper) OTL(PIDE_504.ProgManualReq) OTL(PIDE_504_RESET) ,XIO(PIDE_504.ProgOper) MOV(FCV_504_SP_Standby_AR,PIDE_504.SPOper) ] ];
   22: XIO(PIDE_504_FRONT_END_CONTROL)XIC(PIDE_504_MODE)[MOV(PT_603.PV,PIDE_504.PV) MOV(PT_603.EuMin,PIDE_504.PVEUMin) MOV(PT_603.EuMax,PIDE_504.PVEUMax) MOV(PIDE_504_COLDBOX_PGAIN,PIDE_504.PGain) MOV(PIDE_504_COLDBOX_IGAIN,PIDE_504.IGain) MOV(100,PIDE_504.SPHLimit) MOV(-2,PIDE_504.SPLLimit) ,ONS(PIDE_504_PVCHANGE2) [XIC(PIDE_504.ProgOper) OTL(PIDE_504.ProgManualReq) OTL(PIDE_504_RESET) ,XIO(PIDE_504.ProgOper) MOV(FCV_504_SP_Standby,PIDE_504.SPOper) ] ];
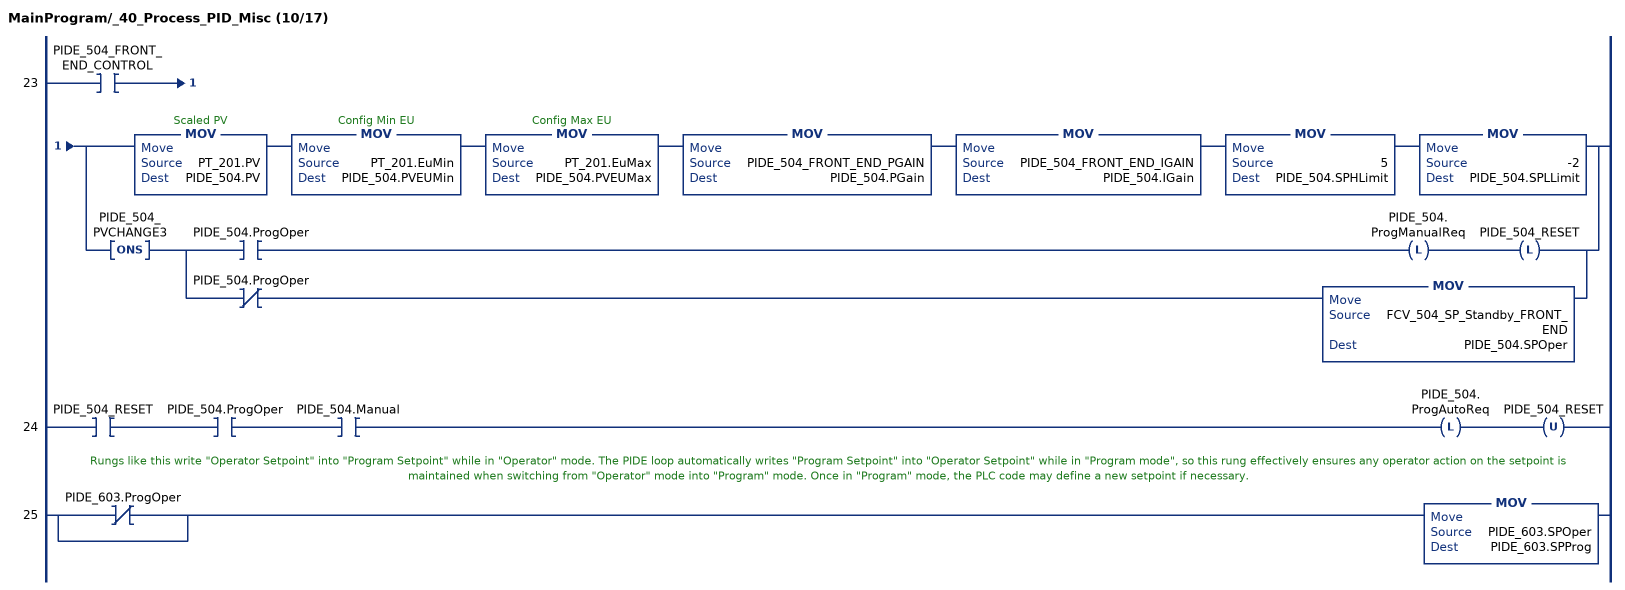
   23: XIC(PIDE_504_FRONT_END_CONTROL)[MOV(PT_201.PV,PIDE_504.PV) MOV(PT_201.EuMin,PIDE_504.PVEUMin) MOV(PT_201.EuMax,PIDE_504.PVEUMax) MOV(PIDE_504_FRONT_END_PGAIN,PIDE_504.PGain) MOV(PIDE_504_FRONT_END_IGAIN,PIDE_504.IGain) MOV(5,PIDE_504.SPHLimit) MOV(-2,PIDE_504.SPLLimit) ,ONS(PIDE_504_PVCHANGE3) [XIC(PIDE_504.ProgOper) OTL(PIDE_504.ProgManualReq) OTL(PIDE_504_RESET) ,XIO(PIDE_504.ProgOper) MOV(FCV_504_SP_Standby_FRONT_END,PIDE_504.SPOper) ] ];
   24: XIC(PIDE_504_RESET)XIC(PIDE_504.ProgOper)XIC(PIDE_504.Manual)OTL(PIDE_504.ProgAutoReq)OTU(PIDE_504_RESET);
   // Rungs like this write "Operator Setpoint" into "Program Setpoint" while in "Operator" mode. The PIDE loop automatically writes "Program Setpoint" into "Operator Setpoint" while in "Program mode", so this rung effectively ensures any operator action on the setpoint is maintained when switching from "Operator" mode into "Program" mode. Once in "Program" mode, the PLC code may define a new setpoint if necessary.
   25: [XIO(PIDE_603.ProgOper) ,]MOV(PIDE_603.SPOper,PIDE_603.SPProg);
